// TwinCAT 3 PLC project mfx_bsm
// ProgramVersion: 3.1.4026.11
// libraries:
//   LCLS General, * (SLAC)
//   lcls-twincat-math, * (SLAC - LCLS)
//   lcls-twincat-motion, * (SLAC)
//   Tc2_EtherCAT, * (Beckhoff Automation GmbH)
//   Tc2_Standard, * (Beckhoff Automation GmbH)
//   Tc2_System, * (Beckhoff Automation GmbH)
//   TcUnit, * (www.tcunit.org)
// project tree:
//   DUTs/ E_DataCollectionSequenceStep.TcDUT
//   GVLs/ Constants.TcGVL
//   ITFs/ I_ResetSequence.TcIO, I_SystemCalibration.TcIO, I_TriggerManager.TcIO
//   / PlcTask.TcTTO, UnitTestTask.TcTTO
//   POUs/ FB_DataCollectionSequence.TcPOU, FB_ResetSequence.TcPOU, FB_SystemCalibration.TcPOU, FB_SystemCalibrationUserInput.TcPOU, FB_TriggerManager.TcPOU, F_GetTimeSinceLastExternalTrigger.TcPOU, Main.TcPOU
//   Test/ FB_DataCollectionSequence_Test.TcPOU, FB_SystemCalibration_Test.TcPOU, PRG_TEST.TcPOU
//   Test/Test doubles/ FB_ResetSequenceTestDouble.TcPOU, FB_SystemCalibrationTestDouble.TcPOU, FB_TriggerManagerTestDouble.TcPOU
// real-time tasks:
//   TASK PlcTask: cycle T#10ms, priority 20, ADS port 350
//   TASK UnitTestTask: cycle T#10ms, priority 1, ADS port 351
// motion (NC):
//   TASK NC-Task 1 SAF: cycle T#2ms, priority 4, ADS port 501
//   TASK NC-Task 1 SVB: cycle T#10ms, priority 8, ADS port 511
//   AXIS ScanningAxisXLinear (id 1)
//     OtherSettings: AllowMotionCmdToSlave=true
//     encoder EncType=1
//     drive DrvType=5
//       Analog: TorqueSetpointScale=10, ScaleFactorActTorque=0.1
//     controller CtrType=1
//       CtrPara: PriorControlFactor=1
//         Observer: BandWidth=20
//   AXIS ScanningAxisXRotation (id 2)
//     OtherSettings: AllowMotionCmdToSlave=true
//     encoder EncType=1
//     drive DrvType=5
//       Analog: TorqueSetpointScale=10, ScaleFactorActTorque=0.1
//     controller CtrType=1
//       CtrPara: PriorControlFactor=1
//         Observer: BandWidth=20
//   AXIS ScanningAxisYLinear (id 3)
//     OtherSettings: AllowMotionCmdToSlave=true
//     encoder EncType=1
//     drive DrvType=5
//       Analog: TorqueSetpointScale=10, ScaleFactorActTorque=0.1
//     controller CtrType=1
//       CtrPara: PriorControlFactor=1
//         Observer: BandWidth=20
//   AXIS ScanningAxisZLinear (id 4)
//     OtherSettings: AllowMotionCmdToSlave=true
//     encoder EncType=1
//     drive DrvType=5
//       Analog: TorqueSetpointScale=10, ScaleFactorActTorque=0.1
//     controller CtrType=1
//       CtrPara: PriorControlFactor=1
//         Observer: BandWidth=20
//   AXIS SampleAxisURotation (id 5)
//     OtherSettings: AllowMotionCmdToSlave=true
//     encoder EncType=1
//     drive DrvType=5
//       Analog: TorqueSetpointScale=10, ScaleFactorActTorque=0.1
//     controller CtrType=1
//       CtrPara: PriorControlFactor=1
//         Observer: BandWidth=20
//   AXIS SampleAxisVRotation (id 6)
//     OtherSettings: AllowMotionCmdToSlave=true
//     encoder EncType=1
//     drive DrvType=5
//       Analog: TorqueSetpointScale=10, ScaleFactorActTorque=0.1
//     controller CtrType=1
//       CtrPara: PriorControlFactor=1
//         Observer: BandWidth=20
//   AXIS GonioAxisLinearX (id 7)
//     OtherSettings: AllowMotionCmdToSlave=true
//     encoder EncType=1
//     drive DrvType=5
//       Analog: TorqueSetpointScale=10, ScaleFactorActTorque=0.1
//     controller CtrType=1
//       CtrPara: PriorControlFactor=1
//         Observer: BandWidth=20
//   AXIS GonioAxisLinearY (id 8)
//     OtherSettings: AllowMotionCmdToSlave=true
//     encoder EncType=1
//     drive DrvType=5
//       Analog: TorqueSetpointScale=10, ScaleFactorActTorque=0.1
//     controller CtrType=1
//       CtrPara: PriorControlFactor=1
//         Observer: BandWidth=20
//   AXIS GonioAxisLinearZ (id 9)
//     OtherSettings: AllowMotionCmdToSlave=true
//     encoder EncType=1
//     drive DrvType=5
//       Analog: TorqueSetpointScale=10, ScaleFactorActTorque=0.1
//     controller CtrType=1
//       CtrPara: PriorControlFactor=1
//         Observer: BandWidth=20
//   AXIS OnAxisLinearX (id 10)
//     OtherSettings: AllowMotionCmdToSlave=true
//     encoder EncType=1
//     drive DrvType=5
//       Analog: TorqueSetpointScale=10, ScaleFactorActTorque=0.1
//     controller CtrType=1
//       CtrPara: PriorControlFactor=1
//         Observer: BandWidth=20
//   AXIS OnAxisLinearY (id 11)
//     OtherSettings: AllowMotionCmdToSlave=true
//     encoder EncType=1
//     drive DrvType=5
//       Analog: TorqueSetpointScale=10, ScaleFactorActTorque=0.1
//     controller CtrType=1
//       CtrPara: PriorControlFactor=1
//         Observer: BandWidth=20
//   AXIS OnAxisLinearZ (id 12)
//     OtherSettings: AllowMotionCmdToSlave=true
//     encoder EncType=1
//     drive DrvType=5
//       Analog: TorqueSetpointScale=10, ScaleFactorActTorque=0.1
//     controller CtrType=1
//       CtrPara: PriorControlFactor=1
//         Observer: BandWidth=20
//   AXIS OnAxisRotationPitch (id 13)
//     OtherSettings: AllowMotionCmdToSlave=true
//     encoder EncType=1
//     drive DrvType=5
//       Analog: TorqueSetpointScale=10, ScaleFactorActTorque=0.1
//     controller CtrType=1
//       CtrPara: PriorControlFactor=1
//         Observer: BandWidth=20
//   AXIS OnAxisRotationYaw (id 14)
//     OtherSettings: AllowMotionCmdToSlave=true
//     encoder EncType=1
//     drive DrvType=5
//       Analog: TorqueSetpointScale=10, ScaleFactorActTorque=0.1
//     controller CtrType=1
//       CtrPara: PriorControlFactor=1
//         Observer: BandWidth=20
//   AXIS CapillaryAxisLinearX (id 15)
//     OtherSettings: AllowMotionCmdToSlave=true
//     encoder EncType=1
//     drive DrvType=5
//       Analog: TorqueSetpointScale=10, ScaleFactorActTorque=0.1
//     controller CtrType=1
//       CtrPara: PriorControlFactor=1
//         Observer: BandWidth=20
//   AXIS CapillaryAxisLinearY (id 16)
//     OtherSettings: AllowMotionCmdToSlave=true
//     encoder EncType=1
//     drive DrvType=5
//       Analog: TorqueSetpointScale=10, ScaleFactorActTorque=0.1
//     controller CtrType=1
//       CtrPara: PriorControlFactor=1
//         Observer: BandWidth=20
//   AXIS CapillaryAxisLinearZ (id 17)
//     OtherSettings: AllowMotionCmdToSlave=true
//     encoder EncType=1
//     drive DrvType=5
//       Analog: TorqueSetpointScale=10, ScaleFactorActTorque=0.1
//     controller CtrType=1
//       CtrPara: PriorControlFactor=1
//         Observer: BandWidth=20
//   AXIS CapillaryAxisRotationPitch (id 18)
//     OtherSettings: AllowMotionCmdToSlave=true
//     encoder EncType=1
//     drive DrvType=5
//       Analog: TorqueSetpointScale=10, ScaleFactorActTorque=0.1
//     controller CtrType=1
//       CtrPara: PriorControlFactor=1
//         Observer: BandWidth=20
// I/O:
//   DEVICE E-Bus (EtherCAT), AmsNetId 199.4.42.250.2.1
//     CX5240BusCoupler (EK1200) [EK1200-5000 EtherCAT Power supply (2A E-Bus)]
//       EL7062_AB_CD-SCXR-SCYL (EL7062) [EL7062-0000 2Ch. Stepper motor output stage (48V, 3A)]
//       Term 3 (EL1252-0050) [EL1252-0050 2Ch. Fast Dig. Input 5V, 1µs, DC Latch]

CONFIGURATION mfx_bsm
    RESOURCE PLC ON TwinCAT3
        TASK PlcTask(INTERVAL := T#10ms, PRIORITY := 20);
        TASK UnitTestTask(INTERVAL := T#10ms, PRIORITY := 1);
        PROGRAM Main WITH PlcTask : Main;
        PROGRAM PRG_TEST WITH UnitTestTask : PRG_TEST;
    END_RESOURCE
END_CONFIGURATION

// ---- DUTs/E_DataCollectionSequenceStep.TcDUT
{attribute 'qualified_only'}
{attribute 'strict'}
{attribute 'to_string'}
TYPE E_DataCollectionSequenceStep :
(
    WaitingForStart := 0,
    // starting positions are all determined by the system calibration result.
    // "SetToStartingStep" button to put the machine in WaitingForInitialTrigger step
    // Query reset system sequence to check that we are indeed fully reset, then we start waiting for initial trigger.
    // When we are waiting for initial trigger, we have an ADS variable that can be queried so the HMI/User knows we are ready to start
    // We need the starting direction to move in and we need to know what the total number of triggers should be
    WaitingForInitialTrigger, // We have to be at the starting x angle, starting z position, starting y position, and starting x position.
    CalculateTimeToNextPoint, // We have a configured number of pulses until we need to be at the first point
    AccelerateToScanningSpeed, // We have a configured acceleration
    OperateAtScanningSpeedMakingMinuteAdjustments,
    GoToNextRow,
    WaitingForTriggerToStartNewRow, // We have to be at the new starting x angle, new starting z position, new starting y position, and new starting x position.
    //CalculateTimeToNextPoint, // We have a configured number of pulses until we need to be at the first point
    //AccelerateToScanningSpeed, // We have a configured acceleration
    //OperateAtScanningSpeedMakingMinuteAdjustments,
    //GoToNextRow,
    Error,
    Done
);
END_TYPE

// ---- GVLs/Constants.TcGVL
{attribute 'qualified_only'}
VAR_GLOBAL CONSTANT
    nGRID_SCAN_POINT_WINDOW_MIN : INT := 0;
    nGRID_SCAN_POINT_WINDOW_MAX : INT := 10;
END_VAR

// ---- ITFs/I_ResetSequence.TcIO
INTERFACE I_ResetSequence

METHOD IsReset : BOOL
END_METHOD

END_INTERFACE

// ---- ITFs/I_SystemCalibration.TcIO
INTERFACE I_SystemCalibration


METHOD PUBLIC ClearLowerLeft
END_METHOD


METHOD PUBLIC ClearLowerRight
END_METHOD


METHOD PUBLIC ClearUpperLeft
END_METHOD


METHOD PUBLIC ClearUpperRight
END_METHOD


METHOD IsCalibrated : BOOL
END_METHOD


METHOD Save
VAR_INPUT
    nWindow : INT;
    fRotationStartAngle : LREAL;
    fRotationStopAngle : LREAL;
    fOscillationVelocity : LREAL;
    fOscillationRange : LREAL;
    nNumberOfRows : INT;
END_VAR
VAR_OUTPUT
    bError : BOOL;
    sErrorString : T_MaxString;
END_VAR
END_METHOD


METHOD PUBLIC SetLowerLeft
VAR_INPUT
    x : LREAL; // [um]
    y : LREAL; // [um]
    z : LREAL; // [um]
END_VAR
END_METHOD


METHOD PUBLIC SetLowerRight
VAR_INPUT
    z : LREAL; // [um]
    x : LREAL; // [um]
    y : LREAL; // [um]
END_VAR
END_METHOD


METHOD PUBLIC SetUpperLeft
VAR_INPUT
    z : LREAL; // [um]
    x : LREAL; // [um]
    y : LREAL; // [um]
END_VAR
END_METHOD


METHOD PUBLIC SetUpperRight
VAR_INPUT
    z : LREAL; // [um]
    x : LREAL; // [um]
    y : LREAL; // [um]
END_VAR
END_METHOD

END_INTERFACE

// ---- ITFs/I_TriggerManager.TcIO
INTERFACE I_TriggerManager

METHOD GetAndResetTrigger
VAR_OUTPUT
    bLatchDetected : BOOL;
    nLatchTime_ns : ULINT; // [ns]
END_VAR
END_METHOD

END_INTERFACE

// ---- POUs/Main.TcPOU

PROGRAM Main
VAR
    fbSystemCalibration : FB_SystemCalibration(nWindowMin := 2,
                                               nWindowMax := 5,
                                               fRotationStartAngleMin := 0.0,
                                               fRotationStartAngleMax  := 90.0,
                                               fRotationStopAngleMin := 0.0,
                                               fRotationStopAngleMax := 90.0,
                                               fOscillationVelocityMin := 10.0,
                                               fOscillationVelocityMax := 45,
                                               fOscillationRangeMin := 20.0,
                                               fOscillationRangeMax := 30.0,
                                               nNumberOfRowsMin := 1,
                                               nNumberOfRowsMax := 6);
    fbSystemCalibrationUserInput : FB_SystemCalibrationUserInput(iSystemCalibration := fbSystemCalibration);
    fbResetSequence : FB_ResetSequence;
    fbTriggerManager : FB_TriggerManager;

    fbDataCollectionSequence : FB_DataCollectionSequence(iSystemCalibration := fbSystemCalibration,
                                                         iResetSequence := fbResetSequence,
                                                         iTriggerManager := fbTriggerManager);

    M1 : ST_MotionStage;
    fbScanningAxisXLinear : FB_MotionStage;
    M2 : ST_MotionStage;
    fbScanningAxisXRotation : FB_MotionStage;
    M3 : ST_MotionStage;
    fbScanningAxisYLinear : FB_MotionStage;
    M4 : ST_MotionStage;
    fbScanningAxisZLinear : FB_MotionStage;

    M5 : ST_MotionStage;
    fbSampleAxisURotation : FB_MotionStage;
    M6 : ST_MotionStage;
    fbSampleAxisVRotation : FB_MotionStage;
    M7 : ST_MotionStage;
    fbGonioAxisLinearX : FB_MotionStage;
    M8 : ST_MotionStage;
    fbGonioAxisLinearY : FB_MotionStage;
    M9 : ST_MotionStage;
    fbGonioAxisLinearZ : FB_MotionStage;
    M10 : ST_MotionStage;
    fbOnAxisLinearX : FB_MotionStage;
    M11 : ST_MotionStage;
    fbOnAxisLinearY : FB_MotionStage;
    M12 : ST_MotionStage;
    fbOnAxisLinearZ : FB_MotionStage;
    M13 : ST_MotionStage;
    fbOnAxisRotationPitch : FB_MotionStage;
    M14 : ST_MotionStage;
    fbOnAxisRotationYaw : FB_MotionStage;
    M15 : ST_MotionStage;
    fbCapillaryAxisLinearX : FB_MotionStage;
    M16 : ST_MotionStage;
    fbCapillaryAxisLinearY : FB_MotionStage;
    M17 : ST_MotionStage;
    fbCapillaryAxisLinearZ : FB_MotionStage;
    M18 : ST_MotionStage;
    fbCapillaryAxisRotationPitch : FB_MotionStage;
END_VAR


fbTriggerManager();

fbSystemCalibrationUserInput();

fbResetSequence();

fbDataCollectionSequence();

IF fbDataCollectionSequence.IsRunningSequence() THEN
    M1.bExecute := FALSE;
    M2.bExecute := FALSE;
    M3.bExecute := FALSE;
    M4.bExecute := FALSE;
    M5.bExecute := FALSE;
    M6.bExecute := FALSE;
    M7.bExecute := FALSE;
    M8.bExecute := FALSE;
    M9.bExecute := FALSE;
    M10.bExecute := FALSE;
    M11.bExecute := FALSE;
    M12.bExecute := FALSE;
    M13.bExecute := FALSE;
    M14.bExecute := FALSE;
    M15.bExecute := FALSE;
    M16.bExecute := FALSE;
    M17.bExecute := FALSE;
    M18.bExecute := FALSE;
END_IF

fbScanningAxisXLinear(stMotionStage := M1);
fbScanningAxisXRotation(stMotionStage := M2);
fbScanningAxisYLinear(stMotionStage := M3);
fbScanningAxisZLinear(stMotionStage := M4);
fbSampleAxisURotation(stMotionStage := M5);
fbSampleAxisVRotation(stMotionStage := M6);
fbGonioAxisLinearX(stMotionStage := M7);
fbGonioAxisLinearY(stMotionStage := M8);
fbGonioAxisLinearZ(stMotionStage := M9);
fbOnAxisLinearX(stMotionStage := M10);
fbOnAxisLinearY(stMotionStage := M11);
fbOnAxisLinearZ(stMotionStage := M12);
fbOnAxisRotationPitch(stMotionStage := M13);
fbOnAxisRotationYaw(stMotionStage := M14);
fbCapillaryAxisLinearX(stMotionStage := M15);
fbCapillaryAxisLinearY(stMotionStage := M16);
fbCapillaryAxisLinearZ(stMotionStage := M17);
fbCapillaryAxisRotationPitch(stMotionStage := M18);

END_PROGRAM

// ---- POUs/FB_SystemCalibration.TcPOU

{attribute 'no_explicit_call' := 'Do not call this POU directly'}
FUNCTION_BLOCK FB_SystemCalibration IMPLEMENTS I_SystemCalibration
VAR
    fbUpperRight : FB_Vec3; // [um]
    bUpperRightCalibrated : BOOL;
    fbUpperLeft : FB_Vec3; // [um]
    bUpperLeftCalibrated : BOOL;
    fbLowerRight : FB_Vec3; // [um]
    bLowerRightCalibrated : BOOL;
    fbLowerLeft : FB_Vec3; // [um]
    bLowerLeftCalibrated : BOOL;

    nWindowMin : INT;
    nWindowMax : INT;
    fRotationStartAngleMin : LREAL; // [°]
    fRotationStartAngleMax : LREAL; // [°]
    fRotationStopAngleMin : LREAL; // [°]
    fRotationStopAngleMax : LREAL; // [°]
    fOscillationVelocityMin : LREAL; // [°/s]
    fOscillationVelocityMax : LREAL; // [°/s]
    fOscillationRangeMin : LREAL; // [°]
    fOscillationRangeMax : LREAL; // [°]
    nNumberOfRowsMin : INT;
    nNumberOfRowsMax : INT;
END_VAR


METHOD PUBLIC ClearLowerLeft

bLowerLeftCalibrated := FALSE;
END_METHOD


METHOD PUBLIC ClearLowerRight

bLowerRightCalibrated := FALSE;
END_METHOD


METHOD PUBLIC ClearUpperLeft

bUpperLeftCalibrated := FALSE;
END_METHOD


METHOD PUBLIC ClearUpperRight

bUpperRightCalibrated := FALSE;
END_METHOD

//FB_Init is always available implicitly and it is used primarily for initialization.
//The return value is not evaluated. For a specific influence, you can also declare the
//methods explicitly and provide additional code there with the standard initialization
//code. You can evaluate the return value.
METHOD FB_Init: BOOL
VAR_INPUT
    bInitRetains: BOOL; // TRUE: the retain variables are initialized (reset warm / reset cold)
    bInCopyCode: BOOL;  // TRUE: the instance will be copied to the copy code afterward (online change)

    nWindowMin : INT;
    nWindowMax : INT;
    fRotationStartAngleMin : LREAL; // [°]
    fRotationStartAngleMax : LREAL; // [°]
    fRotationStopAngleMin : LREAL; // [°]
    fRotationStopAngleMax : LREAL; // [°]
    fOscillationVelocityMin : LREAL; // [°/s]
    fOscillationVelocityMax : LREAL; // [°/s]
    fOscillationRangeMin : LREAL; // [°]
    fOscillationRangeMax : LREAL; // [°]
    nNumberOfRowsMin : INT;
    nNumberOfRowsMax : INT;
END_VAR

THIS^.nWindowMin := nWindowMin;
THIS^.nWindowMax := nWindowMax;
THIS^.fRotationStartAngleMin := fRotationStartAngleMin;
THIS^.fRotationStartAngleMax := fRotationStartAngleMax;
THIS^.fRotationStopAngleMin := fRotationStopAngleMin;
THIS^.fRotationStopAngleMax := fRotationStopAngleMax;
THIS^.fOscillationVelocityMin := fOscillationVelocityMin;
THIS^.fOscillationVelocityMax := fOscillationVelocityMax;
THIS^.fOscillationRangeMin := fOscillationRangeMin;
THIS^.fOscillationRangeMax := fOscillationRangeMax;
THIS^.nNumberOfRowsMin := nNumberOfRowsMin;
THIS^.nNumberOfRowsMax := nNumberOfRowsMax;
END_METHOD


METHOD IsCalibrated : BOOL

IsCalibrated := bUpperRightCalibrated AND
                bUpperLeftCalibrated AND
                bLowerRightCalibrated AND
                bLowerLeftCalibrated;
END_METHOD


METHOD PRIVATE IsWithinRange_INT : BOOL
VAR_INPUT
    Value : INT;
    Maximum : INT;
    Minimum : INT;
    Inclusive : BOOL := TRUE;
END_VAR

IF Inclusive THEN
    IsWithinRange_INT := Value <= Maximum AND Value >= Minimum;
ELSE
    IsWithinRange_INT := Value < Maximum AND Value > Minimum;
END_IF
END_METHOD


METHOD PRIVATE IsWithinRange_LREAL : BOOL
VAR_INPUT
    Value : LREAL;
    Maximum : LREAL;
    Minimum : LREAL;
    Inclusive : BOOL := TRUE;
END_VAR

IF Inclusive THEN
    IsWithinRange_LREAL := Value <= Maximum AND Value >= Minimum;
ELSE
    IsWithinRange_LREAL := Value < Maximum AND Value > Minimum;
END_IF
END_METHOD


METHOD PUBLIC Save
VAR_INPUT
    nWindow : INT;
    fRotationStartAngle : LREAL;
    fRotationStopAngle : LREAL;
    fOscillationVelocity : LREAL;
    fOscillationRange : LREAL;
    nNumberOfRows : INT;
END_VAR
VAR_OUTPUT
    bError : BOOL;
    sErrorString : T_MaxString;
END_VAR

IF NOT IsCalibrated() THEN
    bError := TRUE;
    sErrorString := 'Can$'t save grid scan points. System is not calibrated';
    RETURN;
END_IF

IF NOT IsWithinRange_INT(Value := nWindow, Maximum := nWindowMax, Minimum := nWindowMin) THEN
    bError := TRUE;
    sErrorString := 'Can$'t save grid scan points. Window number is out of range';
    RETURN;
END_IF

IF NOT IsWithinRange_LREAL(Value := fRotationStartAngle, Maximum := fRotationStartAngleMax, Minimum := fRotationStartAngleMin) THEN
    bError := TRUE;
    sErrorString := 'Can$'t save grid scan points. Rotation start angle is out of range';
    RETURN;
END_IF

IF NOT IsWithinRange_LREAL(Value := fRotationStopAngle, Maximum := fRotationStopAngleMax, Minimum := fRotationStopAngleMin) THEN
    bError := TRUE;
    sErrorString := 'Can$'t save grid scan points. Rotation stop angle is out of range';
    RETURN;
END_IF

IF NOT IsWithinRange_LREAL(Value := fOscillationVelocity, Maximum := fOscillationVelocityMax, Minimum := fOscillationVelocityMin) THEN
    bError := TRUE;
    sErrorString := 'Can$'t save grid scan points. Oscillation velocity is out of range';
    RETURN;
END_IF

IF NOT IsWithinRange_LREAL(Value := fOscillationRange, Maximum := fOscillationRangeMax, Minimum := fOscillationRangeMin) THEN
    bError := TRUE;
    sErrorString := 'Can$'t save grid scan points. Oscillation range is out of range';
    RETURN;
END_IF

IF NOT IsWithinRange_INT(Value := nNumberOfRows, Maximum := nNumberOfRowsMax, Minimum := nNumberOfRowsMin) THEN
    bError := TRUE;
    sErrorString := 'Can$'t save grid scan points. Number of rows is out of range';
    RETURN;
END_IF
END_METHOD


METHOD PUBLIC SetLowerLeft
VAR_INPUT
    x : LREAL; // [um]
    y : LREAL; // [um]
    z : LREAL; // [um]
END_VAR

fbLowerLeft.x := x;
fbLowerLeft.y := y;
fbLowerLeft.z := z;
bLowerLeftCalibrated := TRUE;
END_METHOD


METHOD PUBLIC SetLowerRight
VAR_INPUT
    z : LREAL; // [um]
    x : LREAL; // [um]
    y : LREAL; // [um]
END_VAR

fbLowerRight.x := x;
fbLowerRight.y := y;
fbLowerRight.z := z;
bLowerRightCalibrated := TRUE;
END_METHOD


METHOD PUBLIC SetUpperLeft
VAR_INPUT
    z : LREAL; // [um]
    x : LREAL; // [um]
    y : LREAL; // [um]
END_VAR

fbUpperLeft.x := x;
fbUpperLeft.y := y;
fbUpperLeft.z := z;
bUpperLeftCalibrated := TRUE;
END_METHOD


METHOD PUBLIC SetUpperRight
VAR_INPUT
    z : LREAL; // [um]
    x : LREAL; // [um]
    y : LREAL; // [um]
END_VAR

fbUpperRight.x := x;
fbUpperRight.y := y;
fbUpperRight.z := z;
bUpperRightCalibrated := TRUE;
END_METHOD

END_FUNCTION_BLOCK

// ---- POUs/FB_SystemCalibrationUserInput.TcPOU

FUNCTION_BLOCK FB_SystemCalibrationUserInput
VAR
    iSystemCalibration : I_SystemCalibration;

    // Inputs from UI
    {attribute 'pytmc' := '
        pv: nWindow
        io: io
    '}
    nWindow : INT;
    {attribute 'pytmc' := '
        pv: fRotationStartAngle
        io: io
    '}
    fRotationStartAngle : LREAL;
    {attribute 'pytmc' := '
        pv: fRotationStopAngle
        io: io
    '}
    fRotationStopAngle : LREAL;
    {attribute 'pytmc' := '
        pv: fOscillationVelocity
        io: io
    '}
    fOscillationVelocity : LREAL;
    {attribute 'pytmc' := '
        pv: fOscillationRange
        io: io
    '}
    fOscillationRange : LREAL;
    {attribute 'pytmc' := '
        pv: nNumberOfRows
        io: io
    '}
    nNumberOfRows : INT;
    {attribute 'pytmc' := '
        pv: bSaveCommand
        io: io
    '}
    bSaveCommand : BOOL;

    {attribute 'pytmc' := '
        pv: bSaveUpperRight
        io: io
    '}
    bSaveUpperRight : BOOL;
    {attribute 'pytmc' := '
        pv: fUpperRightX
        io: io
    '}
    fUpperRightX : LREAL;
    {attribute 'pytmc' := '
        pv: fUpperRightY
        io: io
    '}
    fUpperRightY : LREAL;
    {attribute 'pytmc' := '
        pv: fUpperRightZ
        io: io
    '}
    fUpperRightZ : LREAL;

    {attribute 'pytmc' := '
        pv: bSaveUpperLeft
        io: io
    '}
    bSaveUpperLeft : BOOL;
    {attribute 'pytmc' := '
        pv: fUpperLeftX
        io: io
    '}
    fUpperLeftX : LREAL;
    {attribute 'pytmc' := '
        pv: fUpperLeftY
        io: io
    '}
    fUpperLeftY : LREAL;
    {attribute 'pytmc' := '
        pv: fUpperLeftZ
        io: io
    '}
    fUpperLeftZ : LREAL;

    {attribute 'pytmc' := '
        pv: bSaveLowerRight
        io: io
    '}
    bSaveLowerRight : BOOL;
    {attribute 'pytmc' := '
        pv: fLowerRightX
        io: io
    '}
    fLowerRightX : LREAL;
    {attribute 'pytmc' := '
        pv: fLowerRightY
        io: io
    '}
    fLowerRightY : LREAL;
    {attribute 'pytmc' := '
        pv: fLowerLeftZ
        io: io
    '}
    fLowerRightZ : LREAL;

    {attribute 'pytmc' := '
        pv: bSaveLowerLeft
        io: io
    '}
    bSaveLowerLeft : BOOL;
    {attribute 'pytmc' := '
        pv: fLowerLeftX
        io: io
    '}
    fLowerLeftX : LREAL;
    {attribute 'pytmc' := '
        pv: fLowerLeftY
        io: io
    '}
    fLowerLeftY : LREAL;
    {attribute 'pytmc' := '
        pv: fLowerLeftZ
        io: io
    '}
    fLowerLeftZ : LREAL;

    {attribute 'pytmc' := '
        pv: bClearAll
        io: io
    '}
    bClearAll : BOOL;
    {attribute 'pytmc' := '
        pv: bClearUpperRight
        io: io
    '}
    bClearUpperRight : BOOL;
    {attribute 'pytmc' := '
        pv: bClearUpperLeft
        io: io
    '}
    bClearUpperLeft : BOOL;
    {attribute 'pytmc' := '
        pv: bClearLowerRight
        io: io
    '}
    bClearLowerRight : BOOL;
    {attribute 'pytmc' := '
        pv: bClearLowerLeft
        io: io
    '}
    bClearLowerLeft : BOOL;

    // Outputs to UI
    {attribute 'pytmc' := '
        pv: bError
        io: i
    '}
    bError : BOOL;
    {attribute 'pytmc' := '
        pv: sErrorString
        io: i
    '}
    sErrorString : T_MaxString;
END_VAR


IF bSaveCommand THEN
    bSaveCommand := FALSE;

    iSystemCalibration.Save(nWindow := nWindow,
                            fRotationStartAngle := fRotationStartAngle,
                            fRotationStopAngle := fRotationStopAngle,
                            fOscillationVelocity := fOscillationVelocity,
                            fOscillationRange := fOscillationRange,
                            nNumberOfRows := nNumberOfRows,
                            bError => bError,
                            sErrorString => sErrorString
    );

    IF bError THEN
        GVL_Logger.fbRootLogger(sMsg := CONCAT('Error attempting system calibration save command: ', sErrorString),
                                eSevr := TcEventSeverity.Error,
                                eSubsystem := E_Subsystem.MOTION
        );
    END_IF
END_IF

IF bSaveUpperRight THEN
    bSaveUpperRight := FALSE;

    iSystemCalibration.SetUpperRight(x := fUpperRightX,
                                     y := fUpperRightY,
                                     z := fUpperRightZ
    );
END_IF

IF bSaveUpperLeft THEN
    bSaveUpperLeft := FALSE;

    iSystemCalibration.SetUpperLeft(x := fUpperLeftX,
                                    y := fUpperLeftY,
                                    z := fUpperLeftZ
    );
END_IF

IF bSaveLowerRight THEN
    bSaveLowerRight := FALSE;

    iSystemCalibration.SetLowerRight(x := fLowerRightX,
                                     y := fLowerRightY,
                                     z := fLowerRightZ
    );
END_IF

IF bSaveLowerLeft THEN
    bSaveLowerLeft := FALSE;

    iSystemCalibration.SetLowerLeft(x := fLowerLeftX,
                                    y := fLowerLeftY,
                                    z := fLowerLeftZ
    );
END_IF

IF bClearAll THEN
    bClearAll := FALSE;

    bClearUpperRight := TRUE;
    bClearUpperLeft := TRUE;
    bClearLowerRight := TRUE;
    bClearLowerRight := TRUE;
END_IF

IF bClearUpperRight THEN
    bClearUpperRight := FALSE;

    iSystemCalibration.ClearUpperRight();
END_IF

IF bClearUpperLeft THEN
    bClearUpperLeft := FALSE;

    iSystemCalibration.ClearUpperLeft();
END_IF

IF bClearLowerRight THEN
    bClearLowerRight := FALSE;

    iSystemCalibration.ClearLowerRight();
END_IF

IF bClearLowerLeft THEN
    bClearLowerLeft := FALSE;

    iSystemCalibration.ClearLowerLeft();
END_IF


//FB_Init is always available implicitly and it is used primarily for initialization.
//The return value is not evaluated. For a specific influence, you can also declare the
//methods explicitly and provide additional code there with the standard initialization
//code. You can evaluate the return value.
METHOD FB_Init: BOOL
VAR_INPUT
    bInitRetains: BOOL; // TRUE: the retain variables are initialized (reset warm / reset cold)
    bInCopyCode: BOOL;  // TRUE: the instance will be copied to the copy code afterward (online change)

    iSystemCalibration : I_SystemCalibration;
END_VAR

THIS^.iSystemCalibration := iSystemCalibration;
END_METHOD

END_FUNCTION_BLOCK

// ---- POUs/FB_ResetSequence.TcPOU

FUNCTION_BLOCK FB_ResetSequence IMPLEMENTS I_ResetSequence
VAR

END_VAR

{warning 'Add method implementation '}
METHOD IsReset : BOOL
END_METHOD

END_FUNCTION_BLOCK

// ---- POUs/FB_TriggerManager.TcPOU
FUNCTION_BLOCK FB_TriggerManager IMPLEMENTS I_TriggerManager
VAR
    nEL1252LatchPos AT %I* : ULINT;
    nEL1252LatchPosPreviousCycle : ULINT;
    bNewLatchPending : BOOL;
END_VAR


IF nEL1252LatchPos <> nEL1252LatchPosPreviousCycle THEN
    bNewLatchPending := TRUE;
END_IF
nEL1252LatchPosPreviousCycle := nEL1252LatchPos;

{warning 'Add method implementation '}
METHOD GetAndResetTrigger
VAR_OUTPUT
    bLatchDetected	: BOOL;
    (* [ns]*)
    nLatchTime_ns	: ULINT;
END_VAR

bLatchDetected := bNewLatchPending;

nLatchTime_ns := nEL1252LatchPos;

bNewLatchPending := FALSE;
END_METHOD

END_FUNCTION_BLOCK

// ---- POUs/FB_DataCollectionSequence.TcPOU

FUNCTION_BLOCK FB_DataCollectionSequence
VAR
    iSystemCalibration : I_SystemCalibration;
    iResetSequence : I_ResetSequence;
    iTriggerManager : I_TriggerManager;

    eSequence : E_DataCollectionSequenceStep;
END_VAR


// Run our sequence here

CASE eSequence OF
    E_DataCollectionSequenceStep.WaitingForStart :
        // Do nothing

    E_DataCollectionSequenceStep.WaitingForInitialTrigger :

    E_DataCollectionSequenceStep.CalculateTimeToNextPoint :

    E_DataCollectionSequenceStep.AccelerateToScanningSpeed :

    E_DataCollectionSequenceStep.OperateAtScanningSpeedMakingMinuteAdjustments :

    E_DataCollectionSequenceStep.GoToNextRow :

    E_DataCollectionSequenceStep.WaitingForTriggerToStartNewRow :

    E_DataCollectionSequenceStep.Error :
        // Do nothing
    E_DataCollectionSequenceStep.Done :
        // Do nothing
END_CASE

//FB_Init is always available implicitly and it is used primarily for initialization.
//The return value is not evaluated. For a specific influence, you can also declare the
//methods explicitly and provide additional code there with the standard initialization
//code. You can evaluate the return value.
METHOD FB_Init: BOOL
VAR_INPUT
    bInitRetains: BOOL; // TRUE: the retain variables are initialized (reset warm / reset cold)
    bInCopyCode: BOOL;  // TRUE: the instance will be copied to the copy code afterward (online change)
    iSystemCalibration : I_SystemCalibration;
    iResetSequence : I_ResetSequence;
    iTriggerManager : I_TriggerManager;
END_VAR
THIS^.iSystemCalibration := iSystemCalibration;
THIS^.iResetSequence := iResetSequence;
THIS^.iTriggerManager := iTriggerManager;
END_METHOD

METHOD PRIVATE GetDataCollectionSequenceStep : E_DataCollectionSequenceStep
GetDataCollectionSequenceStep := THIS^.eSequence;
END_METHOD

METHOD PUBLIC IsRunningSequence : BOOL
IsRunningSequence := (GetDataCollectionSequenceStep() <> E_DataCollectionSequenceStep.WaitingForStart) AND
                     (GetDataCollectionSequenceStep() <> E_DataCollectionSequenceStep.Error) AND
                     (GetDataCollectionSequenceStep() <> E_DataCollectionSequenceStep.Done);
END_METHOD


METHOD PUBLIC Start
VAR_OUTPUT
    bError : BOOL;
    sErrorString : T_MaxString;
END_VAR

IF NOT iSystemCalibration.IsCalibrated() THEN
    bError := TRUE;
    sErrorString := 'Can$'t start data collection sequence. System is not calibrated';
    RETURN;
END_IF

IF NOT iResetSequence.IsReset() THEN
    bError := TRUE;
    sErrorString := 'Can$'t start data collection sequence. System is not reset';
    RETURN;
END_IF

IF eSequence <> E_DataCollectionSequenceStep.WaitingForStart AND eSequence <> E_DataCollectionSequenceStep.Error THEN
    bError := TRUE;
    sErrorString := 'Can$'t start data collection sequence. System is already running data collection sequence';
    RETURN;
END_IF

// Start the sequence
eSequence := E_DataCollectionSequenceStep.WaitingForInitialTrigger;
END_METHOD

END_FUNCTION_BLOCK

// ---- Test/PRG_TEST.TcPOU

PROGRAM PRG_TEST
VAR
    fbDataCollectionSequence_Test : FB_DataCollectionSequence_Test;
    fbSystemCalibration_Test : FB_SystemCalibration_Test;
END_VAR


TcUnit.RUN();

END_PROGRAM

// ---- Test/FB_DataCollectionSequence_Test.TcPOU

FUNCTION_BLOCK FB_DataCollectionSequence_Test EXTENDS FB_TestSuite
VAR
END_VAR


GivenThatSystemIsNotCalibratedDontAllowToStartSequence();


METHOD PRIVATE GivenThatSystemIsNotCalibratedDontAllowToStartSequence
VAR
    fbSystemCalibrationTestDouble : FB_SystemCalibrationTestDouble;
    fbResetSequenceTestDouble : FB_ResetSequenceTestDouble;
    fbTriggerManagerTestDouble : FB_TriggerManagerTestDouble;
    fbDataCollectionSequence : FB_DataCollectionSequence(iSystemCalibration := fbSystemCalibrationTestDouble,
                                                         iResetSequence := fbResetSequenceTestDouble,
                                                         iTriggerManager := fbTriggerManagerTestDouble);

    bErrorReturn : BOOL;
    sErrorStringReturn : T_MaxString;
END_VAR

TEST(__POUNAME());

fbResetSequenceTestDouble.SetIsReset(bIsReset := TRUE);
fbSystemCalibrationTestDouble.SetIsCalibrated(bIsCalibrated := FALSE);


fbDataCollectionSequence.Start(bError => bErrorReturn,
                               sErrorString => sErrorStringReturn);

AssertTrue(Condition := bErrorReturn,
           Message := 'Expected error');

AssertTrue(Condition := sErrorStringReturn <> '',
           Message := 'Expected non-empty string');

TEST_FINISHED();
END_METHOD

END_FUNCTION_BLOCK

// ---- Test/Test doubles/FB_SystemCalibrationTestDouble.TcPOU

FUNCTION_BLOCK FB_SystemCalibrationTestDouble IMPLEMENTS I_SystemCalibration
VAR
    bIsCalibrated : BOOL;
END_VAR


METHOD ClearLowerLeft
END_METHOD


METHOD ClearLowerRight
END_METHOD


METHOD ClearUpperLeft
END_METHOD


METHOD ClearUpperRight
END_METHOD


METHOD IsCalibrated : BOOL
IsCalibrated := THIS^.bIsCalibrated;
END_METHOD


METHOD Save
VAR_INPUT
    nWindow	: INT;
    fRotationStartAngle	: LREAL;
    fRotationStopAngle	: LREAL;
    fOscillationVelocity	: LREAL;
    fOscillationRange	: LREAL;
    nNumberOfRows	: INT;
END_VAR
VAR_OUTPUT
    bError	: BOOL;
    sErrorString	: T_MaxString;
END_VAR
END_METHOD

METHOD SetIsCalibrated : BOOL
VAR_INPUT
    bIsCalibrated : BOOL;
END_VAR
THIS^.bIsCalibrated := bIsCalibrated;
END_METHOD


METHOD SetLowerLeft
VAR_INPUT
    (* [um]*)
    x	: LREAL;
    (* [um]*)
    y	: LREAL;
    (* [um]*)
    z	: LREAL;
END_VAR
END_METHOD


METHOD SetLowerRight
VAR_INPUT
    (* [um]*)
    z	: LREAL;
    (* [um]*)
    x	: LREAL;
    (* [um]*)
    y	: LREAL;
END_VAR
END_METHOD


METHOD SetUpperLeft
VAR_INPUT
    (* [um]*)
    z	: LREAL;
    (* [um]*)
    x	: LREAL;
    (* [um]*)
    y	: LREAL;
END_VAR
END_METHOD


METHOD SetUpperRight
VAR_INPUT
    (* [um]*)
    z	: LREAL;
    (* [um]*)
    x	: LREAL;
    (* [um]*)
    y	: LREAL;
END_VAR
END_METHOD

END_FUNCTION_BLOCK

// ---- Test/Test doubles/FB_ResetSequenceTestDouble.TcPOU
FUNCTION_BLOCK FB_ResetSequenceTestDouble IMPLEMENTS I_ResetSequence
VAR
    bIsResetted : BOOL;
END_VAR

METHOD IsReset : BOOL
IsReset := THIS^.bIsResetted;
END_METHOD

METHOD PUBLIC SetIsReset
VAR_INPUT
    bIsReset : BOOL;
END_VAR
THIS^.bIsResetted := bIsReset;
END_METHOD

END_FUNCTION_BLOCK

// ---- Test/Test doubles/FB_TriggerManagerTestDouble.TcPOU
FUNCTION_BLOCK FB_TriggerManagerTestDouble IMPLEMENTS I_TriggerManager
VAR_INPUT
END_VAR
VAR_OUTPUT
END_VAR
VAR
END_VAR

{warning 'Add method implementation '}
METHOD GetAndResetTrigger
VAR_OUTPUT
    bLatchDetected	: BOOL;
    (* [ns]*)
    nLatchTime_ns	: ULINT;
END_VAR
END_METHOD

END_FUNCTION_BLOCK

// ---- Test/FB_SystemCalibration_Test.TcPOU

FUNCTION_BLOCK FB_SystemCalibration_Test EXTENDS FB_TestSuite
VAR
END_VAR


GivenThatAllFourCornersHaveBeenSetExpectTheSystemToBeCalibrated();
GivenThatAllThreeCornersHaveBeenSetExpectTheSystemNotToBeCalibrated();
GivenThatStartAngleIsNotWithinRangeDontAcceptSave();
GivenThatSystemIsCalibratedAndClearOneIsSetExpectTheSystemNotToBeCalibrated();
GivenThatSystemIsNotCalibratedDontAcceptSave();


METHOD PRIVATE AllPrerequisitesFulfilledAcceptSave
VAR
    fbSystemCalibration : FB_SystemCalibration(nWindowMin := 2,
                                         nWindowMax := 5,
                                         fRotationStartAngleMin := 0.0,
                                         fRotationStartAngleMax  := 90.0,
                                         fRotationStopAngleMin := 0.0,
                                         fRotationStopAngleMax := 90.0,
                                         fOscillationVelocityMin := 10.0,
                                         fOscillationVelocityMax := 45,
                                         fOscillationRangeMin := 20.0,
                                         fOscillationRangeMax := 30.0,
                                         nNumberOfRowsMin := 1,
                                         nNumberOfRowsMax := 6);

    bErrorReturn : BOOL;
    sErrorStringReturn : T_MaxString;

    nWindow : INT;
    fRotationStartAngle : LREAL;
    fRotationStopAngle : LREAL;
    fOscillationVelocity : LREAL;
    fOscillationRange : LREAL;
    nNumberOfRows : INT;
END_VAR

TEST(__POUNAME());

// Test setup
GetNominalValues(fbSystemCalibration := fbSystemCalibration,
                 nWindow => nWindow,
                 fRotationStartAngle => fRotationStartAngle,
                 fRotationStopAngle => fRotationStopAngle,
                 fOscillationVelocity => fOscillationVelocity,
                 fOscillationRange => fOscillationRange,
                 nNumberOfRows => nNumberOfRows);

fbSystemCalibration.Save(nWindow := nWindow,
                      fRotationStartAngle := fRotationStartAngle,
                      fRotationStopAngle := fRotationStopAngle,
                      fOscillationVelocity := fOscillationVelocity,
                      fOscillationRange := fOscillationRange,
                      nNumberOfRows := nNumberOfRows,
                      bError => bErrorReturn,
                      sErrorString => sErrorStringReturn);

AssertFalse(Condition := bErrorReturn,
            Message := 'Expected save to be successful');

AssertEquals_STRING(Expected := '',
                    Actual := sErrorStringReturn,
                    Message := 'Expected string to be empty');

TEST_FINISHED();
END_METHOD

METHOD PRIVATE GetNominalValues
VAR_IN_OUT
    fbSystemCalibration : FB_SystemCalibration;
END_VAR
VAR_OUTPUT
    nWindow : INT;
    fRotationStartAngle : LREAL;
    fRotationStopAngle : LREAL;
    fOscillationVelocity : LREAL;
    fOscillationRange : LREAL;
    nNumberOfRows : INT;
END_VAR

nWindow := 3;
fRotationStartAngle := 0.0;
fRotationStopAngle := 90.0;
fOscillationVelocity := 10.0;
fOscillationRange := 20.0;
nNumberOfRows := 6;

fbSystemCalibration.SetLowerLeft(1, 1, 1);
fbSystemCalibration.SetLowerRight(1, 1, 1);
fbSystemCalibration.SetUpperLeft(1, 1, 1);
fbSystemCalibration.SetUpperRight(1, 1, 1);
END_METHOD


METHOD PRIVATE GivenThatAllFourCornersHaveBeenSetExpectTheSystemToBeCalibrated
VAR
    fbSystemCalibration : FB_SystemCalibration(nWindowMin := 2,
                                         nWindowMax := 5,
                                         fRotationStartAngleMin := 0.0,
                                         fRotationStartAngleMax  := 90.0,
                                         fRotationStopAngleMin := 0.0,
                                         fRotationStopAngleMax := 90.0,
                                         fOscillationVelocityMin := 10.0,
                                         fOscillationVelocityMax := 45,
                                         fOscillationRangeMin := 20.0,
                                         fOscillationRangeMax := 30.0,
                                         nNumberOfRowsMin := 1,
                                         nNumberOfRowsMax := 6);
END_VAR

TEST(__POUNAME());

fbSystemCalibration.SetLowerLeft(z := 1.0,
                                 x := 1.0,
                                 y := 1.0);

fbSystemCalibration.SetLowerRight(z := 1.0,
                                 x := 1.0,
                                 y := 1.0);

fbSystemCalibration.SetUpperLeft(z := 1.0,
                                 x := 1.0,
                                 y := 1.0);

fbSystemCalibration.SetUpperRight(z := 1.0,
                                 x := 1.0,
                                 y := 1.0);

AssertTrue(fbSystemCalibration.IsCalibrated(),
           Message := 'Expected system to be calibrated');

TEST_FINISHED();
END_METHOD


METHOD PRIVATE GivenThatAllThreeCornersHaveBeenSetExpectTheSystemNotToBeCalibrated
VAR
    fbSystemCalibration : FB_SystemCalibration(nWindowMin := 2,
                                         nWindowMax := 5,
                                         fRotationStartAngleMin := 0.0,
                                         fRotationStartAngleMax  := 90.0,
                                         fRotationStopAngleMin := 0.0,
                                         fRotationStopAngleMax := 90.0,
                                         fOscillationVelocityMin := 10.0,
                                         fOscillationVelocityMax := 45,
                                         fOscillationRangeMin := 20.0,
                                         fOscillationRangeMax := 30.0,
                                         nNumberOfRowsMin := 1,
                                         nNumberOfRowsMax := 6);
END_VAR

TEST(__POUNAME());

fbSystemCalibration.SetLowerLeft(z := 1.0,
                                 x := 1.0,
                                 y := 1.0);

fbSystemCalibration.SetLowerRight(z := 1.0,
                                 x := 1.0,
                                 y := 1.0);

fbSystemCalibration.SetUpperLeft(z := 1.0,
                                 x := 1.0,
                                 y := 1.0);

AssertFalse(fbSystemCalibration.IsCalibrated(),
            Message := 'Expected system to not be calibrated');

TEST_FINISHED();
END_METHOD


METHOD PRIVATE GivenThatStartAngleIsNotWithinRangeDontAcceptSave
VAR
    fbSystemCalibration : FB_SystemCalibration(nWindowMin := 2,
                                         nWindowMax := 5,
                                         fRotationStartAngleMin := 0.0,
                                         fRotationStartAngleMax  := 90.0,
                                         fRotationStopAngleMin := 0.0,
                                         fRotationStopAngleMax := 90.0,
                                         fOscillationVelocityMin := 10.0,
                                         fOscillationVelocityMax := 45,
                                         fOscillationRangeMin := 20.0,
                                         fOscillationRangeMax := 30.0,
                                         nNumberOfRowsMin := 1,
                                         nNumberOfRowsMax := 6);

    bErrorReturn : BOOL;
    sErrorStringReturn : T_MaxString;

    nWindow : INT;
    fRotationStartAngle : LREAL;
    fRotationStopAngle : LREAL;
    fOscillationVelocity : LREAL;
    fOscillationRange : LREAL;
    nNumberOfRows : INT;
END_VAR

TEST(__POUNAME());

// Test setup
GetNominalValues(fbSystemCalibration := fbSystemCalibration,
                 nWindow => nWindow,
                 fRotationStartAngle => fRotationStartAngle,
                 fRotationStopAngle => fRotationStopAngle,
                 fOscillationVelocity => fOscillationVelocity,
                 fOscillationRange => fOscillationRange,
                 nNumberOfRows => nNumberOfRows);

fRotationStartAngle := 155.0;

fbSystemCalibration.Save(nWindow := nWindow,
                      fRotationStartAngle := fRotationStartAngle,
                      fRotationStopAngle := fRotationStopAngle,
                      fOscillationVelocity := fOscillationVelocity,
                      fOscillationRange := fOscillationRange,
                      nNumberOfRows := nNumberOfRows,
                      bError => bErrorReturn,
                      sErrorString => sErrorStringReturn);

AssertTrue(Condition := bErrorReturn,
           Message := 'Expected save to not be successful');

AssertTrue(Condition := sErrorStringReturn <> '',
           Message := 'Expected string to not be empty');

TEST_FINISHED();
END_METHOD


METHOD PRIVATE GivenThatSystemIsCalibratedAndClearOneIsSetExpectTheSystemNotToBeCalibrated
VAR
    fbSystemCalibration : FB_SystemCalibration(nWindowMin := 2,
                                         nWindowMax := 5,
                                         fRotationStartAngleMin := 0.0,
                                         fRotationStartAngleMax  := 90.0,
                                         fRotationStopAngleMin := 0.0,
                                         fRotationStopAngleMax := 90.0,
                                         fOscillationVelocityMin := 10.0,
                                         fOscillationVelocityMax := 45,
                                         fOscillationRangeMin := 20.0,
                                         fOscillationRangeMax := 30.0,
                                         nNumberOfRowsMin := 1,
                                         nNumberOfRowsMax := 6);
END_VAR

TEST(__POUNAME());

fbSystemCalibration.SetLowerLeft(z := 1.0,
                                 x := 1.0,
                                 y := 1.0);

fbSystemCalibration.SetLowerRight(z := 1.0,
                                 x := 1.0,
                                 y := 1.0);

fbSystemCalibration.SetUpperLeft(z := 1.0,
                                 x := 1.0,
                                 y := 1.0);

fbSystemCalibration.SetUpperRight(z := 1.0,
                                 x := 1.0,
                                 y := 1.0);

fbSystemCalibration.ClearLowerLeft();

AssertFalse(fbSystemCalibration.IsCalibrated(),
            Message := 'Expected system to not be calibrated');

TEST_FINISHED();
END_METHOD


METHOD PRIVATE GivenThatSystemIsNotCalibratedDontAcceptSave
VAR
    fbSystemCalibration : FB_SystemCalibration(nWindowMin := 2,
                                         nWindowMax := 5,
                                         fRotationStartAngleMin := 0.0,
                                         fRotationStartAngleMax  := 90.0,
                                         fRotationStopAngleMin := 0.0,
                                         fRotationStopAngleMax := 90.0,
                                         fOscillationVelocityMin := 10.0,
                                         fOscillationVelocityMax := 45,
                                         fOscillationRangeMin := 20.0,
                                         fOscillationRangeMax := 30.0,
                                         nNumberOfRowsMin := 1,
                                         nNumberOfRowsMax := 6);

    bErrorReturn : BOOL;
    sErrorStringReturn : T_MaxString;

    nWindow : INT;
    fRotationStartAngle : LREAL;
    fRotationStopAngle : LREAL;
    fOscillationVelocity : LREAL;
    fOscillationRange : LREAL;
    nNumberOfRows : INT;
END_VAR

TEST(__POUNAME());

// Test setup
GetNominalValues(fbSystemCalibration := fbSystemCalibration,
                 nWindow => nWindow,
                 fRotationStartAngle => fRotationStartAngle,
                 fRotationStopAngle => fRotationStopAngle,
                 fOscillationVelocity => fOscillationVelocity,
                 fOscillationRange => fOscillationRange,
                 nNumberOfRows => nNumberOfRows);

fbSystemCalibration.ClearLowerLeft();

AssertFalse(Condition := fbSystemCalibration.IsCalibrated(),
           Message := 'Expected system to not be calibrated in order to run valid test');

fbSystemCalibration.Save(nWindow := nWindow,
                      fRotationStartAngle := fRotationStartAngle,
                      fRotationStopAngle := fRotationStopAngle,
                      fOscillationVelocity := fOscillationVelocity,
                      fOscillationRange := fOscillationRange,
                      nNumberOfRows := nNumberOfRows,
                      bError => bErrorReturn,
                      sErrorString => sErrorStringReturn);

AssertTrue(Condition := bErrorReturn,
           Message := 'Expected save to not be successful');

AssertTrue(Condition := sErrorStringReturn <> '',
           Message := 'Expected string to not be empty');

TEST_FINISHED();
END_METHOD

END_FUNCTION_BLOCK

// ---- POUs/F_GetTimeSinceLastExternalTrigger.TcPOU

FUNCTION F_GetTimeSinceLastExternalTrigger : LREAL // [us]
VAR_INPUT
    LastExternalTriggerTimeLatch : ULINT; // [ns]
END_VAR
VAR
    dcSysTime : ULINT; // [ns]
END_VAR


dcSysTime := F_GetCurDcTickTime64();

IF dcSysTime > LastExternalTriggerTimeLatch THEN
    F_GetTimeSinceLastExternalTrigger := ULINT_TO_LREAL(dcSysTime - LastExternalTriggerTimeLatch) / 1000.0;
ELSE
    F_GetTimeSinceLastExternalTrigger := -ULINT_TO_LREAL(LastExternalTriggerTimeLatch - dcSysTime) / 1000.0;
END_IF

END_FUNCTION
